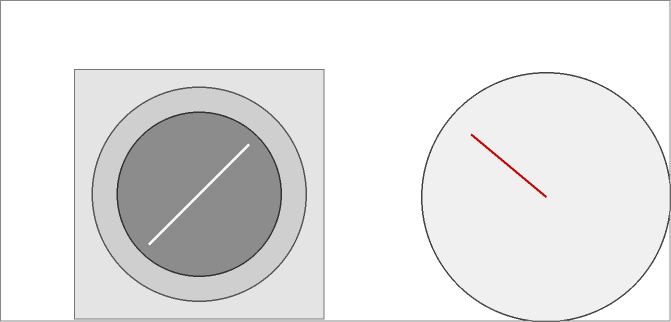
VISUALIZATION Visu_gewicht_en_snelheid  // 671x322
    Meter180 (421,72 250x250), value: GVL.geschrevenSnelheid, style: Meter-Meter180-Gray, scale format: %.1f, scale 0..100
    Potentiometer360 (74,69 250x250), variable: GVL.ladingGewicht, style: Potentiometer-Potentiometer360-Gray, scale format: %.1f, scale 0..100
        p2431819421: Outside
END_VISUALIZATION

(* stored: Version 1.1.0.1, ProductVersion 3.1.4024.12
   Visu Visu_gewicht_en_snelheid: Id {4ee2473c-06f1-407c-bd17-de8ff528ca65} *)
